# EPICS autosave request: iocBoot/ioc13ide_linux/Galil_positions.req
file "CARS_40_motor_positions.req",     P=$(P)
